				Output.SkillOutput[3].Name   :='Block';
	            Output.SkillOutput[3].ID     := 1315 ;	
				Output.SkillOutput[3].Ready  := FALSE ;
				Output.SkillOutput[3].Dummy  := FALSE ; 
	            Output.SkillOutput[3].Done   := FALSE ;
				Output.SkillOutput[3].Busy   := FALSE ;
				Output.SkillOutput[3].ParameterOutput[1].Name := 'TaskID';
				Output.SkillOutput[3].ParameterOutput[1].Dummy:= FALSE;
				Output.SkillOutput[3].ParameterOutput[1].Required:= TRUE ;
				Output.SkillOutput[3].ParameterOutput[1].MinValue:= 1;
				Output.SkillOutput[3].ParameterOutput[1].MaxValue:=30000 ;
				
				// SKILL 4 unblock INTIALISIEREN 
				
				Output.SkillOutput[4].Name   :='Unblock' ;
	            Output.SkillOutput[4].ID     := 1316 ;	
				Output.SkillOutput[4].Ready  := FALSE ;
				Output.SkillOutput[4].Dummy  := FALSE ; 
	            Output.SkillOutput[4].Done   := FALSE ;
				Output.SkillOutput[4].Busy   := FALSE ;
				Output.SkillOutput[4].ParameterOutput[1].Name :=   'TaskID';
				Output.SkillOutput[4].ParameterOutput[1].Dummy:= FALSE;
				Output.SkillOutput[4].ParameterOutput[1].Required:= TRUE ;
				Output.SkillOutput[4].ParameterOutput[1].MinValue:= 1    ;
				Output.SkillOutput[4].ParameterOutput[1].MaxValue:= 30000 ;
				
				// SKILL 5 transport INITIALISIEREN 
				
				Output.SkillOutput[5].Name   :='Transport' ;
	            Output.SkillOutput[5].ID     := 1320 ;	
				Output.SkillOutput[5].Ready  := FALSE ;
				Output.SkillOutput[5].Dummy  := FALSE ; 
	            Output.SkillOutput[5].Done   := FALSE ;
				Output.SkillOutput[5].Busy   := FALSE ;
				Output.SkillOutput[5].ParameterOutput[1].Name := 'TargetPosition X';
				Output.SkillOutput[5].ParameterOutput[1].Dummy:= FALSE;
				Output.SkillOutput[5].ParameterOutput[1].Required:= TRUE ;
				Output.SkillOutput[5].ParameterOutput[1].MinValue:= 0    ;
				Output.SkillOutput[5].ParameterOutput[1].MaxValue:= 4000 ;
				Output.SkillOutput[5].ParameterOutput[2].Name := 'TargetPosition Z';
				Output.SkillOutput[5].ParameterOutput[2].Dummy:= FALSE;
				Output.SkillOutput[5].ParameterOutput[2].Required:= FALSE ;
				Output.SkillOutput[5].ParameterOutput[2].MinValue:= 0.0    ;
				Output.SkillOutput[5].ParameterOutput[2].MaxValue:= 90.0 ;
				Output.SkillOutput[5].ParameterOutput[2].Default:= 0.0; 
				Output.SkillOutput[5].ParameterOutput[3].Name := 'Velocity';
				Output.SkillOutput[5].ParameterOutput[3].Dummy:= FALSE;
				Output.SkillOutput[5].ParameterOutput[3].Required:= FALSE ;
				Output.SkillOutput[5].ParameterOutput[3].MinValue:= 100    ;
				Output.SkillOutput[5].ParameterOutput[3].MaxValue:= 4000 ;
				Output.SkillOutput[5].ParameterOutput[3].Default := 2000;
				Output.SkillOutput[5].ParameterOutput[4].Name := 'Acceleration';
				Output.SkillOutput[5].ParameterOutput[4].Dummy:= FALSE;
				Output.SkillOutput[5].ParameterOutput[4].Required:= FALSE ;
				Output.SkillOutput[5].ParameterOutput[4].MinValue:= 100    ;
				Output.SkillOutput[5].ParameterOutput[4].MaxValue:= 4000 ;
				
				state := 0;
				
			0: // Unreserved 
				IF AwaitingAxisCnt>0 THEN
					AwaitingAxisCnt := AwaitingAxisCnt -1;
					state := 1;				
				END_IF
			
			
	    	1:		// Unreserved
					FOR i := 0 TO SkillCnt DO 
					Output.SkillOutput[i].Ready := FALSE;
					Output.SkillOutput[i].Busy := FALSE;
					Output.SkillOutput[i].Done := FALSE;
					Output.SkillOutput[i].Error := FALSE;
					END_FOR
					
					Output.SkillOutput[1].Ready                    :=TRUE; //reserve
					Output.SkillOutput[0].Ready                    :=TRUE;
					 
	            	             
	
	             	IF Input.SkillInput[1].Execute THEN 
	                
	                	Output.SkillOutput[1].Ready := FALSE ;
						Output.SkillOutput[0].Ready := FALSE ;
						Output.SkillOutput[1].Busy  := TRUE ;
						state:=10 ;
					
					END_IF
					IF Input.SkillInput[0].Execute THEN
	                	Output.SkillOutput[0].Ready := FALSE ;
						Output.SkillOutput[1].Ready := FALSE ;
						Output.SkillOutput[0].Busy  := FALSE ;
						state:=85 ;
	                			FOR i := 1 TO Grpcnt DO
										IF Output.SkillOutput[0].Busy THEN
											state := 1;
											
										END_IF
								END_FOR
						Output.SkillOutput[0].Busy  := TRUE ;
					END_IF
				   
			10:	//Reserve			     	
					IF AwaitingReservationAxis > 0 THEN
						
						//find, which mover is next in line for reservation
						
						MoverNo := AwaitingReservationAxis;
						 
						MoverInfo[AwaitingReservationAxis].blocked := FALSE;
						
						awaitingreservationaxis := 0;
						Nextaxis := F_SetAxInSection(AwaitingReservationAxis -1);
						
						//IF MoverInterface[moverNO].Setpos = WaitingAbsPosition THEN
							state := 12;
						//END_IF
							
	             	//Set mover to reserved in Global Mover Info
						
					
					
	            		MoverInfo[MoverNo].reserved:=TRUE;
						MoverInfo[MoverNo].TaskID	:= REAL_TO_INT (Input.SkillInput[1].ParameterInput[1].Value);
	                
	                	
						Output.SkillOutput[1].Done := TRUE;
						Output.SkillOutput[1].Busy := FALSE;
						Output.SkillOutput[1].Error := FALSE;
						
						
						state:=13 ;
						fbTransport(execute := FALSE, reset := TRUE); 
					END_IF
			13:		//IF NOT MoverInfo[Nextaxis].reserved THEN
					//AwaitingReservationAxis := nextaxis;
					//END_IF


					// internal Block mover next in line
					//MoverInfo[nextaxis].blocked := TRUE;
					
					IF MoverInterface[moverno].Setpos = WaitingAbsPosition	THEN		
						fbTransport( axisno := moverno, execute := TRUE,RequestPosition := F_SetInSection(WaitingAbsPosition + 2* couplegap + 5.0),requestvelo := defaultvelo);
						state := 14;
						
					ELSE
						state := 15;
					END_IF
			14: 
			
				fbTransport( axisno := moverno,RequestPosition := F_SetInSection(WaitingAbsPosition + 2* couplegap + 5.0),requestvelo := defaultvelo);
				IF fbTransport.done THEN
					state := 15;
					fbTransport(reset := TRUE);
				END_IF
		
			15:		//warten bis execute zurückgezogen
					IF NOT(Input.SkillInput[1].Execute) THEN
						Output.SkillOutput[1].Done := FALSE;
						state:=20;
					END_IF
					
					
				 
				 
	  		20:		//Reserved
					IdleTimer(IN := FALSE);
					fbIdleReservedTransport(reset := TRUE);
					state := 21;
			21:
					fbAutoBlock(axno := MoverNo);
					
					IdleTimer(IN := TRUE, PT := T#1000S);
					IF IdleTimer.Q AND (Moverinfo[F_SetAxInSection(Moverno-1)].reserved) THEN
						fbIdleReservedTransport.AxisNo := MoverNo;
						IF NOT (idletempposition = F_SetInSection( Moverinfo[F_SetAxInSection(Moverno+1)].preposition - WaySectionGap - 0.1 - Curvedistance) )THEN
						idletempposition := F_SetInSection( Moverinfo[F_SetAxInSection(Moverno+1)].preposition - WaySectionGap - 0.1 - Curvedistance);
						fbIdleReservedTransport(reset := TRUE);
						END_IF
						IF NOT F_CheckIfInCurve(idletempposition) THEN
								IF Moverinfo[F_SetAxInSection(Moverno+1)].reserved THEN
								fbIdleReservedTransport.RequestPosition := idletempposition;
								ELSE	
								fbIdleReservedTransport.RequestPosition := WaitingAbsPosition - 6 * WaySectionGap - 0.1;
								END_IF
								fbIdleReservedTransport.execute := TRUE;
								curvedistance := 0;
						ELSE
						curvedistance := curvedistance + 10.0;	
						END_IF
					END_IF
					
					fbIdleReservedTransport();
					
					FOR i := 0 TO SkillCnt DO 
					Output.SkillOutput[i].Ready := FALSE;
					Output.SkillOutput[i].Busy := FALSE;
					Output.SkillOutput[i].Done := FALSE;
					Output.SkillOutput[i].Error := FALSE;
					END_FOR
					
					Output.SkillOutput[2].Ready := TRUE;
					Output.SkillOutput[3].Ready := TRUE;
					Output.SkillOutput[5].Ready := TRUE;
					
	              	IF Input.SkillInput[5].Execute THEN 
						fbTransport(reset := TRUE);									   (*in Case of transportation*)
	                    state:=30;	
						Output.SkillOutput[5].Done := FALSE;
						Output.SkillOutput[5].Busy := TRUE;
						FOR i := 0 TO SkillCnt DO 
						Output.SkillOutput[i].Ready := FALSE;
						END_FOR					
					END_IF
	
	             	IF  Input.SkillInput[2].Execute THEN   (*Mover releasing *)
	                    state :=50;
						fbTransport(reset := TRUE);
						Output.SkillOutput[2].Busy := TRUE;
						FOR i := 0 TO SkillCnt DO 
						Output.SkillOutput[i].Ready := FALSE;
						END_FOR	
					END_IF
	
	            	IF Input.SkillInput[3].Execute THEN   (*blocking *)
	                    state:=60;
						fbTransport(reset := TRUE);
						Output.SkillOutput[3].Busy := TRUE;
						FOR i := 0 TO SkillCnt DO 
						Output.SkillOutput[i].Ready := FALSE;
						END_FOR	
				    END_IF		
	
					 
			30:	 //TRANSPORT		
					fbAutoBlock(axno := MoverNo);			
	 				IF Input.SkillInput[5].ParameterInput[4].Value> 0 AND Input.SkillInput[5].ParameterInput[4].Value < nocurvesvelo THEN
					MoverInfo[MoverNo].nocurvestop := TRUE;	
					END_IF
	                
			
			
					fbTransport(
								execute:= TRUE, 
								RequestPosition := Input.SkillInput[5].ParameterInput[1].Value,
								AxisNo:= MoverNo, 
								requestacc := Input.SkillInput[5].ParameterInput[4].Value,
								requestvelo := Input.SkillInput[5].ParameterInput[3].Value,								
								ready=> , 
								error=> , 
								busy=> , 
								done=> 
								);
	
	               IF fbTransport.done THEN             
	               state:=31 ;
				   fbTransport(reset := TRUE);
				   MoverInfo[MoverNo].blocked 	:= TRUE;				   
				   END_IF
				   
				31: 	//überprüfen ob z anforderung
						fbAutoBlock(axno := MoverNo);
						IF Input.SkillInput[5].ParameterInput[2].Value = 0 THEN
							state := 40;
						ELSE state := 32;
						END_IF
				32:		IF 		(1500<Input.SkillInput[5].ParameterInput[1].Value AND (2000+couplegap)>Input.SkillInput[5].ParameterInput[1].Value)
							OR 	(3500<Input.SkillInput[5].ParameterInput[1].Value AND (4000)>Input.SkillInput[5].ParameterInput[1].Value) OR (Input.SkillInput[5].ParameterInput[1].Value<couplegap)
							OR (0.0>Input.SkillInput[5].ParameterInput[2].Value OR 111.0<Input.SkillInput[5].ParameterInput[2].Value)
						THEN // nicht zugelassen!
							state := 41;
							fbAutoBlock(axno := MoverNo);
							Output.SkillOutput[1].done  :=FALSE;
	                    	Output.SkillOutput[2].ready :=FALSE;
	                    	Output.SkillOutput[3].ready :=FALSE;
	                    	Output.SkillOutput[4].ready :=FALSE;
	                    	Output.SkillOutput[5].done  :=FALSE;
							Output.SkillOutput[5].Error := TRUE;
							Output.SkillOutput[5].busy	:= FALSE;
						ELSE
							state := 35;				                   
						END_IF
						
						
						//z-bewegung
				35: 	fbZTransport.execute := TRUE;
						state := 36;
						
						
				36: 
						fbZTransport( zPosition := Input.SkillInput[5].ParameterInput[2].Value, axno := MoverNo);
						IF fbZTransport.done THEN						
							fbAutoBlock(execute := FALSE,axno := MoverNo);
				   			fbAutoBlock(execute := TRUE);
							state := 40;
						END_IF
						
						
				40:	    
						fbAutoBlock(axno := MoverNo,execute := FALSE);
						fbAutoBlock(axno := MoverNo,execute := TRUE);
						
						Output.SkillOutput[5].done  :=TRUE;
						Output.SkillOutput[5].busy	:= FALSE;
						
	                    state:=41;
						
						
				41:		//warten bis execute zurückgezogen
						fbAutoBlock(axno := MoverNo);
						Output.SkillOutput[5].busy	:= FALSE;
						Output.SkillOutput[5].done  :=TRUE;
							IF NOT(Input.SkillInput[5].Execute) THEN
								state:=20 ;
								Output.SkillOutput[5].Done := FALSE;
							END_IF
						
						   
				50:		//Release
							MoverInfo[MoverNo].nocurvestop := FALSE;
	              		 	MoverInfo[MoverNo].reserved := FALSE;
							MoverInfo[MoverNo].blocked := FALSE;
	                       	MoverInfo[MoverNo].TaskID	:= 0;
							MoverNo						:= 0;
							AwaitingAxisCnt := AwaitingAxisCnt +1;
							
						Output.SkillOutput[2].busy := FALSE;
						Output.SkillOutput[2].done := TRUE;
	  					state:=51 ;
						
				51:		//warten bis execute zurückgezogen
						IF NOT(Input.SkillInput[2].Execute) THEN
							state:=0 ;
							Output.SkillOutput[2].Done := FALSE;
						END_IF
						   
						//Block
				60:	  
							
	                        
						MoverInfo[MoverNo].blocked 	:= TRUE;
						  
	                    Output.SkillOutput[3].busy:=FALSE;
						Output.SkillOutput[3].done:=TRUE;
						   
	                    state:=61;
						
				61:		//warten bis execute zurückgezogen
						Output.SkillOutput[3].done:=TRUE;
						IF NOT(Input.SkillInput[3].Execute) THEN
							state:=70 ;
							Output.SkillOutput[3].Done := FALSE;
						END_IF
						   
	            70:		//BLOCKED
						FOR i := 0 TO SkillCnt DO 
						Output.SkillOutput[i].Ready := FALSE;
						Output.SkillOutput[i].Busy := FALSE;
						Output.SkillOutput[i].Done := FALSE;
						Output.SkillOutput[i].Error := FALSE;
						END_FOR			
						Output.SkillOutput[4].Ready := TRUE;
						
						IF Input.SkillInput[4].Execute THEN
							state := 80;
							Output.SkillOutput[4].busy   :=TRUE ;
							Output.SkillOutput[4].Ready := FALSE;
							
						END_IF
	
	
	           	80:         // Unblock;
						MoverInfo[MoverNo].blocked := FALSE;
						MoverInterface[Moverno].Buddyenable := FALSE;
						Output.SkillOutput[4].busy  :=FALSE ;
						Output.SkillOutput[4].Done	:= TRUE;
						
						state := 81;
						
	       		81:     //warten bis execute zurückgezogen
						Output.SkillOutput[4].Done	:= TRUE;
						IF NOT(Input.SkillInput[4].Execute) THEN
							state:=20; 
							Output.SkillOutput[4].Done := FALSE;
						END_IF       
				


				85:		//Initialization
						//IF NOT GVL.ClientExecute THEN
						InitMoverNo := AwaitingReservationAxis;
						state := 86;
						Output.SkillOutput[0].Error := FALSE;
						//END_IF
				86: 	
						state := 87;
						FOR i := 1 TO grpcnt DO
							IF MoverInfo[i].reserved THEN
								state := 86;
							END_IF
						END_FOR
						IF NOT MoverInfo[F_SetAxInSection(grp :=InitMoverNo-1)].reserved THEN
						InitMoverNo := F_SetAxInSection(InitMoverNo-1);
						ELSE
							state := 88;
						END_IF
						
				87: // alle mover unreserved
					IF NOT (AwaitingReservationAxis = 0) THEN
					InitMoverNo := F_SetAxInSection(grp := AwaitingReservationAxis +1);
					state := 88;
					Timeout(IN := FALSE);
					END_IF
					
				88: //OPC COnnection
					//IF NOT GVL.ClientExecute THEN
							AveragedPosition := 0;
							ClientWrite := FALSE;
							FOR i := 1 TO 10 DO Gvl.MeasuredPosition[i] := 0;
								
							END_FOR
								
							GVL.ClientExecute := TRUE;
							GVL.ClientModuleServerUrl 	:= Input.SkillInput[0].ParameterInput[0].StringValue;
							GVL.ClientReadIdentifier	:= Input.SkillInput[0].ParameterInput[1].StringValue;
							GVL.ClientWriteIdentifier 	:= Input.SkillInput[0].ParameterInput[2].StringValue;
							GVL.ClientNamespaceIndex	:= STRING_TO_UINT (Input.SkillInput[0].ParameterInput[3].StringValue);
							GVL.ClientNamespaceUri		:= Input.SkillInput[0].ParameterInput[4].StringValue;
							IF GVL.ClientReadEstablished THEN
								state := 89;
							END_IF
							
							Timeout(IN := TRUE, PT := T#10S);
							IF Timeout.Q THEN
								Timeout(IN := FALSE);
							state := 107;
							Output.SkillOutput[0].Busy := FALSE;
							Output.SkillOutput[0].Error := TRUE;
								
							END_IF
					//END_IF
					
				89: MoverInfo[InitMoverNo].reserved := TRUE;
					fbTransport(execute := TRUE, AxisNo := InitMoverNo,RequestPosition := F_SetInSection(WaitingAbsPosition - 5.5* WaySectionGap), requestvelo := maxvelo);
					IF MoverInterface[InitMoverNo].Targetpos = F_SetInSection(WaitingAbsPosition - 5.5* WaySectionGap) THEN
                  		state := 90;
					END_IF
				90: fbTransport();
					IF fbTransport.done THEN
						state := 91;
						fbTransport(reset := TRUE);
					END_IF
				91:	
					fbTransport(execute := TRUE, AxisNo := InitMoverNo,RequestPosition := WaitingAbsPosition + 2.5* WaySectionGap, requestvelo := initvelo);
					IF MoverInterface[InitMoverNo].Targetpos = WaitingAbsPosition + 2.5* WaySectionGap THEN
                  		state := 92;
					END_IF
					
				
				92: fbTransport(); // erste suche
					IF bInput THEN 
					tempposition := F_SetInSection(ax[InitMoverNo*2].NcToPlc.ModuloActPos );
					fbTransport(execute := FALSE, reset := TRUE);
					state := 95;
					END_IF
					IF fbTransport.done THEN
						IF measuredposition[1] = 0 THEN
							state := 106;
						ELSE
						state := 95;
						END_IF
					END_IF
				
					
				95: IF measuredcycles = measurementCycles THEN
						state  := 100;
					ELSE					
					//in position fahren
					fbTransport(execute := TRUE, AxisNo := InitMoverNo, RequestPosition := F_SetInSection(Tempposition + ((EXPT(-1,measuredcycles)) * 100)),requestvelo := 2000);
					IF NOT bInput AND fbTransport.done THEN
						
					state := 96;
					END_IF
					END_IF
					
				96: //Messung
					fbTransport(execute := TRUE, AxisNo := InitMoverNo, RequestPosition := F_SetInSection(Tempposition - ((EXPT(-1,measuredcycles)) * 300)) ,requestvelo := 50);
					IF bInput THEN
					MeasuredPosition[measuredcycles +1] := ax[2*InitMoverNo].NcToPlc.ModuloActPos;
					measuredcycles := measuredcycles +1;
					fbTransport(execute := FALSE, Reset := TRUE);
					state := 95;
					END_IF
					IF fbTransport.done THEN
						state := 95;
						repeatcounter := repeatcounter + 1;
					END_IF
					IF Repeatcounter > Measurementcycles + 20 THEN
						
							state := 107;
							Output.SkillOutput[0].Busy := FALSE;
							Output.SkillOutput[0].Error := TRUE;
							
					END_IF
					
				100: 
						i := 1;
						state := 103;
				103: 
					IF i <= measurementCycles THEN
						AveragedPosition := AveragedPosition + (EXPT(measurementCycles,-1) * ( measuredposition[i]));
						i := i+1;
					ELSE
						fbTransport(reset := TRUE, execute := FALSE);
						state := 105;
						Timeout(IN := FALSE);
						AveragedPosition := F_SetInSection(AveragedPosition - 33.5);					
					END_IF
				105: 
					fbTransport(execute := TRUE, AxisNo := InitMoverNo, RequestPosition := AveragedPosition);
					IF fbTransport.done THEN
						state := 106;
						Timeout(IN := FALSE);
						fbTransport(reset := TRUE);
					END_IF
				106: 	ClientWrite := TRUE;
						Timeout(IN := TRUE, PT := T#100S);
							IF Timeout.Q THEN
								Timeout(IN := FALSE);
							state := 1070;
							Output.SkillOutput[0].Busy := FALSE;
							Output.SkillOutput[0].Error := TRUE;
								
							END_IF
						IF GVL.ClientDone THEN
						
					 	state := 107;
						OUTput.SkillOutput[0].Done := TRUE;
						OUTput.SkillOutput[0].busy := FALSE; 
					 	END_IF
			    107:	//auf execute zurückziehen warten 
						ClientExecute := FALSE;
						fbTransport(reset := TRUE);
						IF NOT Input.SkillInput[0].Execute THEN
						MoverInfo[InitMoverNo].reserved := FALSE;
						OUTput.SkillOutput[0].Done := FALSE;
						Output.SkillOutput[0].Busy := FALSE;
						state := 1;
						measuredcycles := 0;
						repeatcounter := 0;
						END_IF
					
					 
							  
						
	END_CASE
	
ELSE //SUPPRESSED!
	fbSuppressedTransport(
	surpressall := TRUE,	
	execute:= TRUE, 
	RequestPosition:= MoverInfo[MoverNo].SurpressedPosition, 
	AxisNo:= MoverNo, 
	ready=> , 
	error=> , 
	busy=> , 
	done=> );
	IF fbSuppressedTransport.done THEN
		fbTransport.reset := TRUE;
		MoverInfo[MoverNo].surpressed := FALSE;
				
	END_IF
END_IF

ELSE
	IF restartstate = 2 THEN
		state := 0;
		fbTransport(reset := TRUE);
		restartstate := 3;
		moverno := 0;
	END_IF
END_IF

Output.ConnectionTestOutput := INput.ConnectionTestInput;

END_FUNCTION_BLOCK

// ---- POUs/SkillHandle/FB_Transport.TcPOU
FUNCTION_BLOCK FB_Transport
VAR_INPUT
	execute: BOOL;
	RequestPosition: LREAL;
	AxisNo: INT;
	reset: BOOL;
	requestvelo: LREAL;
	requestacc: LREAL;
	surpressall: BOOL;
	test1: BOOL;
	test2: BOOL;
END_VAR
VAR_OUTPUT
	ready: BOOL;
	error: BOOL;
	busy: BOOL;
	done: BOOL;
END_VAR
VAR
	///FBs
	calculateWaysection: FB_CalculateWaysection;
	checkWaysection: FB_CheckWaysection;
	Clockwise: BOOL;
	TempPreposition: LREAL;
	TempPostposition: LREAL;
	BlockingAxisNo: INT;
	state: INT := 10;
	surpressCheck	: BOOL := FALSE;
	i: INT;
	CatchUp	: BOOL;
END_VAR

IF reset THEN
	state := 10;
	reset := FALSE;
	done := FALSE;
	execute := FALSE;
	calculateWaysection(Execute := FALSE);
	checkWaysection(Execute := FALSE);
END_IF
IF execute THEN 
	done := FALSE;
	busy := TRUE;
	CASE state OF 
	10: // calculate clockwise
			calculateWaysection(
					Clockwise:= TRUE, 
					Startpos:= MoverInterface[AxisNo].Setpos,
					Endpos:= RequestPosition, 
					WaySectionGap:= WaySectionGap, 
					Execute:= TRUE, 
					Prepos=> TempPreposition, 
					Postpos=> TempPostposition, 
					done=> );
			IF calculateWaysection.done THEN state := 15; END_IF
			
	15: // immer nur einer gleichzeitig checken:
		IF Reservingaxis = 0  OR Reservingaxis = AxisNo THEN
			Reservingaxis := AxisNo;
			state := 20;
		END_IF
	20: // check clockwise waysection & reserve if free
			checkWaysection(
							CheckPreposition:= TempPreposition, 
							CheckPostposition:= TempPostposition, 
							CheckMoverNo:= AxisNo , 
							Execute:= TRUE, 
							SectionFree=> , 
							axisblocking=> , 
							done=> );
							
			IF checkWaysection.done THEN
				Reservingaxis := 0;
					IF checkWaysection.SectionFree THEN
						//Section frei -> Reservieren!
							MoverInfo[AxisNo].postposition 	:= TempPostposition;
							MoverInfo[AxisNo].preposition	:= TempPreposition;
							state := 100;
							Clockwise := TRUE;
							
						ELSE
							state := 25;
					END_IF
				
			END_IF
	
	25: // immer nur einer gleichzeitig checken:
		IF Reservingaxis = 0 OR Reservingaxis = AxisNo THEN
			Reservingaxis := AxisNo;
			state := 30;
		END_IF	
	
	30: //calculate counter-clockwise
		calculateWaysection(
					Clockwise:= FALSE, 
					Startpos:= MoverInterface[AxisNo].Setpos,
					Endpos:= RequestPosition, 
					WaySectionGap:= WaySectionGap, 
					Execute:= TRUE, 
					Prepos=> TempPreposition, 
					Postpos=> TempPostposition, 
					done=> );
			IF calculateWaysection.done THEN state := 40; END_IF
	
	40: //check counter-clockwise waysection
		checkWaysection(
							CheckPreposition:= TempPreposition, 
							CheckPostposition:= TempPostposition, 
							CheckMoverNo:= AxisNo , 
							Execute:= TRUE, 
							SectionFree=> , 
							axisblocking=> , 
							done=> );
							
			IF checkWaysection.done THEN
				Reservingaxis := 0;
					IF checkWaysection.SectionFree
						THEN //Section frei -> Reservieren!
							MoverInfo[AxisNo].postposition 	:= TempPostposition;
							MoverInfo[AxisNo].preposition	:= TempPreposition;
							state := 100;
							Clockwise := FALSE;
					ELSE	//section nicht frei
						state := 50;
					END_IF			
			END_IF
	
	50: //Find Out blocking axNo
		BlockingAxisNo := AxisNo -1;
		IF AxisNo = 1 THEN
			BlockingAxisNo := grpcnt;
		END_IF
		state := 60;
	
	60: 		test1 :=F_CheckIfInSection(Position := WaitingAbsPosition - 6 * WaySectionGap, postposition := MoverInterface[AxisNo].Setpos, preposition := F_SetInSection(TempPreposition - WaySectionGap -0.1));
				test2 := F_CheckSurpressedSection(SurpressedPosition := F_SetInSection(TempPreposition - WaySectionGap -0.1), preposition := F_SetInSection(WaitingAbsPosition - 3 * couplegap), postposition := MoverInterface[AxisNo].Setpos);
		IF NOT surpressCheck THEN
			state  := 10;
			surpresscheck := TRUE;
		ELSE
			
				IF 
					NOT MoverInfo[BlockingAxisNo].blocked 
					AND NOT (Moverinfo[axisno].surpressed AND Moverinfo[F_SetAxInSection(axisno +1)].surpressed )    
					AND 	(surpressall OR
							(*  (NOT F_CheckIfInSection(Position:=MoverInterface[blockingaxisno].Targetpos, postposition := WaitingAbsPosition, preposition := F_SetInSection( Waitingabsposition - 6 * (waysectiongap + 0.1))) 
								AND NOT F_CheckSurpressedSection(SurpressedPosition := F_SetInSection(TempPreposition - WaySectionGap -0.1), preposition := F_SetInSection(WaitingAbsPosition - 3 * couplegap), postposition := MoverInterface[AxisNo].Setpos))
							*)
							NOT F_CheckIfInSection(Position := WaitingAbsPosition - 6 * WaySectionGap, postposition := MoverInterface[AxisNo].Setpos, preposition := F_SetInSection(TempPreposition - WaySectionGap -0.2))
							)
						
							// ACHSE Verdrängen
				THEN	MoverInfo[BlockingAxisNo].surpressed := TRUE;
						surpresscheck := FALSE;	
							//verdängungsposition berechnen
							IF NOT (F_CheckIfInCurve (TempPreposition - WaySectionGap -0.2) AND MoverInfo[i].nocurvestop) THEN
							MoverInfo[BlockingAxisNo].SurpressedPosition :=  F_SetInSection(TempPreposition - WaySectionGap -0.2);
							ELSE
								IF F_SetInSection(TempPreposition - WaySectionGap -0.2 ) > 2500 THEN
									// hintere kurve
									MoverInfo[BlockingAxisNo].SurpressedPosition :=  3450;
								ELSE
									//vordere Kurve
									MoverInfo[BlockingAxisNo].SurpressedPosition :=  1450;
								END_IF
							
							END_IF
							
							
							//gegen den uhrzeigersinn ausweichen:
							MoverInfo[BlockingAxisNo].SupressedClockwise := FALSE;
							state := 70; //auf verdrängung warten
					ELSE
							state := 10; //warten/neue Berechnung
							IF (Moverinfo[axisno].surpressed AND Moverinfo[F_SetAxInSection(axisno +1)].surpressed ) THEN
							ADSLOGSTR(ADSLOG_MSGTYPE_HINT, 'trying to surpress all movers! Help!', '');
							state := 10;	
							END_IF
				END_IF
			END_IF
	
	70: 	//Wait untill suppressed movement done
			// Supressed mover Rücken auf
			
			IF  (MoverInfo[AxisNo].preposition - MoverInfo[BlockingAxisNo].postposition ) > (surpressinggap + 600) THEN
				
			
			MoverInfo[AxisNo].preposition 	:= F_SetinSection(MoverInfo[BlockingAxisNo].postposition + surpressinggap);
			MoverInfo[AxisNo].postposition	:= F_SetinSection(MoverInterface[AxisNo].Setpos + waysectiongap);
			MoverInterface[AxisNo].targetpos := F_SetInSection(MoverInfo[BlockingAxisNo].postposition + waysectiongap + surpressinggap);
			CAInterface.MoverInterface[AxisNo].Clockwise := FALSE;
			CatchUp := TRUE;
			ELSE
			CatchUp := FALSE;
			END_IF
			surpresscheck := FALSE;
				
			state := 71;
	71: 	
			// immer nur einer gleichzeitig checken:
			IF Reservingaxis = 0 OR Reservingaxis = AxisNo THEN
				Reservingaxis := AxisNo;
				state := 30;
			END_IF	
	72:
			checkWaysection(
							CheckPreposition:= TempPreposition, 
							CheckPostposition:= TempPostposition, 
							CheckMoverNo:= AxisNo , 
							Execute:= TRUE, 
							SectionFree=> , 
							axisblocking=> , 
							done=> );
			
							
			IF checkWaysection.done THEN
					Reservingaxis := 0;
					IF checkWaysection.SectionFree
						THEN //Section frei -> Reservieren!
							MoverInfo[AxisNo].postposition 	:= TempPostposition;
							MoverInfo[AxisNo].preposition	:= TempPreposition;
							state := 100;
							Clockwise := FALSE;
					ELSE
						state :=71;
					END_IF			
			END_IF
			IF CatchUp THEN
				//reservierten bereich während der fahr freigeben
			IF ((CAInterface.MoverInterface[axisno].Setpos + WaySectionGap)> railLength) THEN //bereich überprüfen
						MoverInfo[AxisNo].postposition := CAInterface.MoverInterface[axisno].Setpos + WaySectionGap -railLength;
			ELSE
						MoverInfo[AxisNo].postposition := CAInterface.MoverInterface[axisno].Setpos + WaySectionGap;
			END_IF
			state := 70;
			END_IF
	
		///BEWEGUNGSAUSFÜHRUNG
	100: 	CAInterface.MoverInterface[AxisNo].Targetpos := RequestPosition;
			CAInterface.MoverInterface[AxisNo].Clockwise := Clockwise;
			CAInterface.MoverInterface[AxisNo].MovementDone := FALSE;
			IF (requestacc > 0.0 AND requestacc < maxacc) THEN
			CAInterface.MoverInterface[AxisNo].Acceleration := requestacc;
			ELSE 
				CAInterface.MoverInterface[AxisNo].Acceleration := defaulacc;
			END_IF
			IF (requestvelo > 0.0 AND requestvelo < maxvelo) THEN
			CAInterface.MoverInterface[AxisNo].Velocity := requestvelo;
			ELSE 
				CAInterface.MoverInterface[AxisNo].Velocity := defaultvelo;
			END_IF
			surpresscheck := FALSE;	
			state := 101;
			
	101:	//reservierten bereich während der fahrt freigeben
			IF Clockwise 
			THEN 
				// Preposition aktualisieren
				
					IF ((CAInterface.MoverInterface[axisno].Setpos - WaySectionGap)< 0.0) THEN //bereich überprüfen
						MoverInfo[AxisNo].preposition := CAInterface.MoverInterface[axisno].Setpos - WaySectionGap +railLength;
					ELSE
						MoverInfo[AxisNo].preposition := CAInterface.MoverInterface[axisno].Setpos - WaySectionGap;
					END_IF
				
			ELSE
				//Postposition aktualisieren
					IF ((CAInterface.MoverInterface[axisno].Setpos + WaySectionGap)> railLength) THEN //bereich überprüfen
						MoverInfo[AxisNo].postposition := CAInterface.MoverInterface[axisno].Setpos + WaySectionGap -railLength;
					ELSE
						MoverInfo[AxisNo].postposition := CAInterface.MoverInterface[axisno].Setpos + WaySectionGap;
					END_IF
			END_IF
			
			//Auf Ende Warten
			IF CAInterface.MoverInterface[AxisNo].MovementDone THEN
		
				state :=  10;
				execute := FALSE;
				busy := FALSE;
				done := TRUE;
					// letztes mal pre/post aktuallisieren
								IF Clockwise 
								THEN 
									// Preposition aktualisieren
									
										IF ((CAInterface.MoverInterface[axisno].Setpos - WaySectionGap)< 0.0) THEN //bereich überprüfen
											MoverInfo[AxisNo].preposition := CAInterface.MoverInterface[axisno].Setpos - WaySectionGap +railLength;
										ELSE
											MoverInfo[AxisNo].preposition := CAInterface.MoverInterface[axisno].Setpos - WaySectionGap;
										END_IF
									
								ELSE
									//Postposition aktualisieren
										IF ((CAInterface.MoverInterface[axisno].Setpos + WaySectionGap)> railLength) THEN //bereich überprüfen
											MoverInfo[AxisNo].postposition := CAInterface.MoverInterface[axisno].Setpos + WaySectionGap -railLength;
										ELSE
											MoverInfo[AxisNo].postposition := CAInterface.MoverInterface[axisno].Setpos + WaySectionGap;
										END_IF
								END_IF
			END_IF
	
	
	
		
	END_CASE
	ELSE state := 10;
END_IF

END_FUNCTION_BLOCK

// ---- POUs/SkillHandle/F_CheckIfInSection.TcPOU
FUNCTION F_CheckIfInSection : BOOL
VAR_INPUT
	Position: LREAL;
	postposition: LREAL;
	preposition: LREAL;
END_VAR
VAR
	InSection: BOOL;
END_VAR


	InSection := FALSE;
		IF postposition>preposition 
		THEN
				//DER RESERVIERTE BEREICH GEHT NICHT ÜBER NULL:	
					
					// gesamter bereich umschlungen?
					IF Position >  preposition AND Position <= PostPosition THEN
						InSection:= TRUE;
					END_IF
				
		ELSE
				//DER RESERVIERTE BEREICH GEHT ÜBER NULL!
				//Bereich 1: 0 bis Postpos:
					// Grenze in Bereich?
					IF((Position>=0.0) AND (Position<=postposition)) 
						THEN 
							InSection:= TRUE;
								
					END_IF
				
				//Bereich 2: Prepos bis 4000
					// Grenze in Bereich?
					IF((Position>=preposition) AND (Position<=raillength)) 
						THEN 
							InSection:= TRUE;
					END_IF	
		END_IF

F_CheckIfInSection := inSection;

END_FUNCTION

// ---- POUs/SkillHandle/F_SetInSection.TcPOU
FUNCTION F_SetInSection : LREAL
VAR_INPUT
	Position: LREAL;
END_VAR
VAR
	output: LREAL;
END_VAR

IF (Position >= raillength) THEN
	output := position -raillength;
ELSE
	IF (Position < 0.0) THEN
		output := position + raillength;
	ELSE
	output := Position;
	END_IF
END_IF
F_SetInSection := output;

END_FUNCTION

// ---- POUs/SkillHandle/F_CheckSurpressedSection.TcPOU
FUNCTION F_CheckSurpressedSection : BOOL
VAR_INPUT
	SurpressedPosition: LREAL;
	postposition: LREAL;
	preposition: LREAL;
END_VAR
VAR
	InSection: BOOL;
END_VAR


	InSection := FALSE;
		IF postposition>preposition 
		THEN
				//DER RESERVIERTE BEREICH GEHT NICHT ÜBER NULL:	
					
					// gesamter bereich umschlungen?
					IF SurpressedPosition >  preposition AND SurpressedPosition <= PostPosition THEN
						InSection:= TRUE;
					END_IF
				
		ELSE
				//DER RESERVIERTE BEREICH GEHT ÜBER NULL!
				//Bereich 1: 0 bis Postpos:
					// Grenze in Bereich?
					IF((SurpressedPosition>=0.0) AND (SurpressedPosition<=postposition)) 
						THEN 
							InSection:= TRUE;
								
					END_IF
				
				//Bereich 2: Prepos bis 4000
					// Grenze in Bereich?
					IF((SurpressedPosition>=preposition) AND (SurpressedPosition<=raillength)) 
						THEN 
							InSection:= TRUE;
					END_IF	
		END_IF

F_CheckSurpressedSection := inSection;

END_FUNCTION

// ---- POUs/SkillHandle/F_SetAxInSection.TcPOU
FUNCTION F_SetAxInSection : INT
VAR_INPUT
	grp: INT := 0;
END_VAR

IF grp < 1 THEN 
	F_SetAxInSection := grp + grpcnt;
ELSE
	IF grp > grpcnt THEN
		F_SetAxInSection := grp  - grpcnt;
	ELSE
		F_SetAxInSection := grp;
	END_IF
END_IF

END_FUNCTION

// ---- POUs/SkillHandle/F_CheckIfInCurve.TcPOU
FUNCTION F_CheckIfInCurve : BOOL
VAR_INPUT
	Position: LREAL;
END_VAR
VAR
	pre1: LREAL := 1490.0;
	end1: LREAL := 2010.0;
	
	pre2: LREAL := 3490.0;
	
	end2: LREAL := 10.0;
END_VAR

F_CheckIfInCurve := F_CheckIfInSection(Position := Position, postposition := end1, preposition := pre1) or F_CheckIfInSection(Position := Position, postposition := end2, preposition := pre2);

END_FUNCTION

// ---- POUs/SkillHandle/FB_AutoBlock.TcPOU
FUNCTION_BLOCK FB_AutoBlock
VAR_INPUT
	execute: BOOL;
	axno: INT;
	blockingtime: TIME := TIME#2s0ms;
END_VAR
VAR
	state: INT := 0;
	fbTimer: TON;
END_VAR

IF NOT Execute THEN
	state := 0;
ELSE
	CASE state OF
		
	0: 
		MoverInfo[axno].blocked := TRUE;
		fbTimer(IN := FALSE);
		fbTimer(IN := TRUE, PT := blockingtime);
		state := 1;
	1:	
		fbTimer();
		IF fbTimer.Q THEN
			MoverInfo[axno].blocked := FALSE;
			execute := FALSE;
			state := 0;
		END_IF
		
	
	
	
	
	END_CASE
END_IF

END_FUNCTION_BLOCK

// ---- POUs/SkillHandle/FB_ZTransport.TcPOU
FUNCTION_BLOCK FB_ZTransport
VAR_INPUT
	execute: BOOL;
	axno: INT;
	zPosition: LREAL;
END_VAR
VAR_OUTPUT
	done: BOOL;
	busy: BOOL;
	error: BOOL;
END_VAR
VAR
	state: INT := 0;
	gap: LREAL;
END_VAR

IF execute THEN
	done	:= FALSE;/// 
	busy := TRUE; ///
	CASE state OF
		
	0: //gap berechnen 12 30 154
		done	:= FALSE;
		busy := TRUE;
		gap := (-0.4123*zPosition)+ zerohightdistance;
		state := 5;
		
	5:	
		CAInterface.MoverInterface[axno].Buddyenable := FALSE;
		IF NOT CAInterface.MoverInterface[axno].Buddyactive THEN
			state := 10;
		END_IF
		
	10: 
		// an CA übergeben
		CAInterface.MoverInterface[axno].Buddygap := gap;
		CAInterface.MoverInterface[axno].Buddyenable := TRUE;
		state := 20;

	20: 
		IF  CAInterface.MoverInterface[axno].Buddyactive THEN
		done := TRUE;
		busy := FALSE;
		execute := FALSE;
		state := 0;
		END_IF
	
	
	
	END_CASE
END_IF

END_FUNCTION_BLOCK

// ---- POUs/SkillHandle/FB_FreeTransport.TcPOU
FUNCTION_BLOCK FB_FreeTransport
VAR_INPUT
	execute: BOOL;
	RequestPosition: LREAL;
	AxisNo: INT;
	reset: BOOL;
END_VAR
VAR_OUTPUT
	ready: BOOL;
	error: BOOL;
	busy: BOOL;
	done: BOOL;
END_VAR
VAR
	///FBs
	calculateWaysection: FB_CalculateWaysection;
	checkWaysection: FB_CheckWaysection;
	Clockwise: BOOL;
	TempPreposition: LREAL;
	TempPostposition: LREAL;
	BlockingAxisNo: INT;
	PostmoverNo: INT;
	state: INT := 10;
	i: INT;
	fbSuppressedTransport: FB_Transport;
END_VAR

//Nummer des nächsten Movers herausfinden
PostmoverNo := F_SetAxInSection( AxisNo +1);


IF NOT Restart THEN

IF NOT MoverInfo[AxisNo].surpressed THEN
	

			IF execute THEN 
				MoverInterface[axisno].Buddyenable:= FALSE;
				done := FALSE;
				busy := TRUE;
				CASE state OF 
				10: // calculate counter-clockwise
						calculateWaysection(
								Clockwise:= FALSE, 
								Startpos:= MoverInterface[AxisNo].Setpos,
								Endpos:= RequestPosition, 
								WaySectionGap:= WaySectionGap, 
								Execute:= TRUE, 
								Prepos=> TempPreposition, 
								Postpos=> TempPostposition, 
								done=> );
						IF calculateWaysection.done THEN state := 15; END_IF
				15:  // immer nur einer gleichzeitig checken:
						IF Reservingaxis = 0 OR Reservingaxis = AxisNo THEN
							Reservingaxis := AxisNo;
							state := 20;
						END_IF
				20: // check counter-clockwise waysection & reserve if free
						checkWaysection(
										CheckPreposition:= TempPreposition, 
										CheckPostposition:= TempPostposition, 
										CheckMoverNo:= AxisNo , 
										Execute:= TRUE, 
										SectionFree=> , 
										axisblocking=> , 
										done=> );
										
						IF checkWaysection.done THEN
							Reservingaxis := 0;
								IF checkWaysection.SectionFree
									THEN //Section frei -> Reservieren!
										MoverInfo[AxisNo].postposition 	:= TempPostposition;
										MoverInfo[AxisNo].preposition	:= TempPreposition;
										state := 100;
										Clockwise := FALSE;
								ELSE state := 25;
								END_IF
							
						END_IF
				
				25: // immer nur einer gleichzeitig checken:
					IF Reservingaxis = 0 OR Reservingaxis = AxisNo THEN
						Reservingaxis := AxisNo;
						state := 30;
					END_IF		
				
				30: //calculate clockwise
					calculateWaysection(
								Clockwise:= TRUE, 
								Startpos:= MoverInterface[AxisNo].Setpos,
								Endpos:= RequestPosition, 
								WaySectionGap:= WaySectionGap, 
								Execute:= TRUE, 
								Prepos=> TempPreposition, 
								Postpos=> TempPostposition, 
								done=> );
						IF calculateWaysection.done THEN state := 40; END_IF
				
				40: //check clockwise waysection
					checkWaysection(
										CheckPreposition:= TempPreposition, 
										CheckPostposition:= TempPostposition, 
										CheckMoverNo:= AxisNo , 
										Execute:= TRUE, 
										SectionFree=> , 
										axisblocking=> , 
										done=> );
										
						IF checkWaysection.done THEN
							Reservingaxis := 0;
								IF checkWaysection.SectionFree
									THEN //Section frei -> Reservieren!
										MoverInfo[AxisNo].postposition 	:= TempPostposition;
										MoverInfo[AxisNo].preposition	:= TempPreposition;
										state := 100;
										Clockwise := TRUE;
								ELSE	//section nicht frei
									state := 50;
								END_IF			
						END_IF
				
						
				50: //Aufschließen
					calculateWaysection(
								Clockwise:= TRUE, 
								Startpos:= MoverInterface[AxisNo].Setpos,
								Endpos:= F_SetInSection(Position := (MoverInfo[PostmoverNo].preposition - WaySectionGap - 0.1)) , 
								WaySectionGap:= WaySectionGap, 
								Execute:= TRUE, 
								Prepos=> TempPreposition, 
								Postpos=> TempPostposition, 
								done=> );
						IF calculateWaysection.done THEN state := 55; END_IF
						
				55:		IF Reservingaxis = 0 THEN
						Reservingaxis := AxisNo;
						state := 60;
						END_IF
						
				60:		
						checkWaysection(
										CheckPreposition:= TempPreposition, 
										CheckPostposition:= TempPostposition, 
										CheckMoverNo:= AxisNo , 
										Execute:= TRUE, 
										SectionFree=> , 
										axisblocking=> , 
										done=> );
										
						IF checkWaysection.done THEN
								Reservingaxis := 0;
								IF checkWaysection.SectionFree
									THEN //Section frei -> Reservieren!
										MoverInfo[AxisNo].postposition 	:= TempPostposition;
										MoverInfo[AxisNo].preposition	:= TempPreposition;
										state := 70;
										Clockwise := TRUE;
								ELSE	//section nicht frei
									state := 10;
								END_IF			
						END_IF
						
				70: 	CAInterface.MoverInterface[AxisNo].Targetpos := F_SetInSection(MoverInfo[PostmoverNo].preposition - WaySectionGap - 0.1);
						CAInterface.MoverInterface[AxisNo].Clockwise := Clockwise;
						CAInterface.MoverInterface[AxisNo].MovementDone := FALSE;
						CAInterface.MoverInterface[AxisNo].Velocity := freevelo;
						CAInterface.MoverInterface[AxisNo].Acceleration := freeacc;
						state := 71;
						
				71:	//reservierten bereich während der fahrt freigeben
						IF Clockwise 
						THEN 
							// Preposition aktualisieren
							
								IF ((CAInterface.MoverInterface[axisno].Setpos - WaySectionGap)< 0.0) THEN //bereich überprüfen
									MoverInfo[AxisNo].preposition := CAInterface.MoverInterface[axisno].Setpos - WaySectionGap +railLength;
								ELSE
									MoverInfo[AxisNo].preposition := CAInterface.MoverInterface[axisno].Setpos - WaySectionGap;
								END_IF
							
						ELSE
							//Postposition aktualisieren
								IF ((CAInterface.MoverInterface[axisno].Setpos + WaySectionGap)> railLength) THEN //bereich überprüfen
									MoverInfo[AxisNo].postposition := CAInterface.MoverInterface[axisno].Setpos + WaySectionGap -railLength;
								ELSE
									MoverInfo[AxisNo].postposition := CAInterface.MoverInterface[axisno].Setpos + WaySectionGap;
								END_IF
						END_IF
						
						//Auf Ende Warten
						IF CAInterface.MoverInterface[AxisNo].MovementDone THEN
					
							state :=  10;
						ELSE
							state := 30;	
						END_IF
				
					///BEWEGUNGSAUSFÜHRUNG
				100: 	CAInterface.MoverInterface[AxisNo].Targetpos := RequestPosition;
						CAInterface.MoverInterface[AxisNo].Clockwise := Clockwise;
						
						CAInterface.MoverInterface[AxisNo].MovementDone := FALSE;
						CAInterface.MoverInterface[AxisNo].Acceleration := freeacc;
						CAInterface.MoverInterface[AxisNo].Velocity := freevelo;
						
						state := 101;
						
				101:	//reservierten bereich während der fahrt freigeben
						IF Clockwise 
						THEN 
							// Preposition aktualisieren
							
								IF ((CAInterface.MoverInterface[axisno].Setpos - WaySectionGap)< 0.0) THEN //bereich überprüfen
									MoverInfo[AxisNo].preposition := CAInterface.MoverInterface[axisno].Setpos - WaySectionGap +railLength;
								ELSE
									MoverInfo[AxisNo].preposition := CAInterface.MoverInterface[axisno].Setpos - WaySectionGap;
								END_IF
							
						ELSE
							//Postposition aktualisieren
								IF ((CAInterface.MoverInterface[axisno].Setpos + WaySectionGap)> railLength) THEN //bereich überprüfen
									MoverInfo[AxisNo].postposition := CAInterface.MoverInterface[axisno].Setpos + WaySectionGap -railLength;
								ELSE
									MoverInfo[AxisNo].postposition := CAInterface.MoverInterface[axisno].Setpos + WaySectionGap;
								END_IF
						END_IF
						
						//Auf Ende Warten
						IF CAInterface.MoverInterface[AxisNo].MovementDone THEN
					
							state :=  10;
							execute := FALSE;
							busy := FALSE;
							done := TRUE;
						END_IF
				
						
				
					
				END_CASE
			END_IF
ELSE //suppressed!
	fbSuppressedTransport(
	surpressall := TRUE,
	execute:= TRUE, 
	RequestPosition:= MoverInfo[AxisNo].SurpressedPosition, 
	AxisNo:= AxisNo, 
	requestvelo := freevelo,
	ready=> , 
	error=> , 
	busy=> , 
	done=> );
	IF fbSuppressedTransport.done THEN
		state := 10;
		MoverInfo[AxisNo].surpressed := FALSE;
				
	END_IF

END_IF

ELSE
	IF restartstate = 3 THEN
		state := 10;
		restartstate := 4;
	END_IF
END_IF

END_FUNCTION_BLOCK

// ---- POUs/SkillHandle/FB_FreeSlotHandle.TcPOU
FUNCTION_BLOCK FB_FreeSlotHandle
VAR_INPUT
	autoexecute: BOOL;
END_VAR
VAR
	fbFreeTransport: ARRAY[1..grpcnt] OF FB_FreeTransport;
	i: INT;
	initdone: BOOL;
	initax: INT := 3;
	minposition: LREAL := 4000.0;
END_VAR

IF NOT initdone AND((MoverInterface[1].MovementDone) AND (MoverInterface[2].MovementDone) AND (MoverInterface[3].MovementDone) ) THEN
	fbFreeTransport[initax](AxisNo := initax, RequestPosition := WaitingAbsPosition,execute := TRUE);
	IF fbFreeTransport[3].done THEN
	autoexecute := TRUE;
	initdone := TRUE;
	END_IF
END_IF

		FOR i := 1 TO grpcnt DO
			IF NOT MoverInfo[i].reserved THEN
				IF NOT (MoverInterface[i].Setpos = WaitingAbsPosition) THEN
					fbFreeTransport[i](AxisNo := i, RequestPosition := WaitingAbsPosition,execute := autoexecute);
					
				ELSE
					fbFreeTransport[i](AxisNo := i, RequestPosition := WaitingAbsPosition,execute := FALSE);
					IF NOT MoverInfo[i].reserved	THEN
					AwaitingReservationAxis := i;
					END_IF
					//MoverInfo[i].blocked := TRUE;
				END_IF
			
					
			END_IF
		 
		END_FOR

END_FUNCTION_BLOCK

// ---- POUs/CAHandle/FB_CAHandle.TcPOU

FUNCTION_BLOCK FB_CAHandle
VAR_OUTPUT
	initdone: BOOL;
	cadone: BOOL;
	reset: BOOL;
END_VAR
VAR
	state: INT := -10;
	resetstate: INT := 2;
	nextstate: INT;
	halt: BOOL;
	forcedisable: BOOL;
	fbpowerall: FB_PowerAll;
	fbresetall: FB_ResetAll;
	fbaddall: FB_AddAllAxes;
	fbremoveall: FB_RemoveAllAxesCA;
	fbhaltall: FB_HaltAll;
	fbCAgrpEnable: MC_GroupEnableCA(calltargetOID);
	fbCAgrpDisable: MC_GroupDisableCA(calltargetOID);
	fbCAgrpReset: MC_GroupResetCA(calltargetOID);
	fbCAgrpStatus: MC_GroupReadStatusCA;
	fbCAgrpError: MC_GroupReadErrorCA;
	fbuncoupleall: FB_UncoupleAll;
	fbCaInterfaceHandle: ARRAY[1..grpcnt] OF FB_CAInterfaceHandle;
	fbCoupleInit: FB_CoupleInit;
	i: UINT;
	targetpos: ARRAY[1..grpcnt] OF LREAL;
	///targetposact: ARRAY[1..grpcnt] OF LREAL;
	movervel: LREAL := 1000;
	railLength: LREAL := 4000;
END_VAR
VAR_INPUT
	executereset: BOOL := TRUE;
	goon: BOOL;
END_VAR


fbpowerall(enable:=TRUE, axes := poweredaxes);
fbCAgrpStatus(AxesGroup:=CAgrp, enable:=TRUE);
fbCAgrpError(AxesGroup:=CAgrp, enable:=TRUE);

IF (fbpowerall.ison ) AND NOT executereset THEN
	CASE state OF
		
		-10: fbCoupleInit(execute := TRUE,startline := WaitingAbsPosition - 100.0 + ax[1].NcToPlc.moduloactturns * 4000);
			IF fbCoupleInit.done THEN
				state := -5;
			END_IF
			
		-5:	fbaddall(Execute:=FALSE);
			fbaddall(Execute:=TRUE);
			
			(* CAinterface.MoverInterface[1].Targetpos := 1000;
			CAinterface.MoverInterface[2].Targetpos := 1500;
			CAinterface.MoverInterface[3].Targetpos := 2000;
			CAinterface.MoverInterface[4].Targetpos := 2500;
			*)
			state := -4;
		-4:	
			fbaddall();
			IF (NOT fbaddall.Busy) THEN
				IF (NOT fbaddall.Error) THEN
					nextstate := -3;
					state := -3; //100
				END_IF
			END_IF
		-3:
			fbCAgrpEnable(AxesGroup:=CAgrp, execute:=FALSE);
			fbCAgrpEnable(AxesGroup:=CAgrp, execute:=TRUE);
			state := -2;
		-2:
			fbCAgrpEnable(AxesGroup:=CAgrp);
			IF (fbCAgrpEnable.Done) THEN
				ADSLOGSTR(ADSLOG_MSGTYPE_HINT, 'XTS Successfully Activated', '');
				nextstate := 0;
				cadone		:= TRUE;
				state := 0;
			END_IF
		0:	// now all axes are in the enabled group, we start with some moves
			FOR i := 1 TO grpcnt DO
			fbCaInterfaceHandle[i](axisno := i, movervel := MoverInterface[i].Velocity, moveracc := MoverInterface[i].Acceleration);	
			END_FOR	
			initdone := TRUE;
			
			
		5:
			fbhaltall(execute:=FALSE);
			fbhaltall(execute:=TRUE);
			state := 6;
		6:	fbhaltall();
			IF (fbhaltall.Done) THEN
				state := 100;
			END_IF
		10:
			fbCAgrpDisable(AxesGroup:=CAgrp, execute:=FALSE);
			fbCAgrpDisable(AxesGroup:=CAgrp, execute:=TRUE);
			state := 11;
		11:	fbCAgrpDisable(AxesGroup:=CAgrp);
			IF (fbCAgrpDisable.Done) THEN
				state := 12;
			END_IF
		12:
			fbremoveall(Execute:=FALSE);
			fbremoveall(Execute:=TRUE);
			state := 13;
		13:	fbremoveall();
			IF (NOT fbremoveall.Busy) THEN
				IF (NOT fbremoveall.Error) THEN
					ADSLOGSTR(ADSLOG_MSGTYPE_HINT, 'All Axes Removed From Group', '');
					nextstate := 14;
					state := 100;
				END_IF
			END_IF
			
		14:	fbresetall(execute:=FALSE);
			fbresetall(execute:=TRUE);
			state := 15;
		15:
			fbresetall();
			IF (NOT fbresetall.Busy) THEN
				IF (NOT fbresetall.Error) THEN
					ADSLOGSTR(ADSLOG_MSGTYPE_HINT, 'All Axes Successfully Reset', '');
					nextstate := -5;
					state := 100;
				END_IF
			END_IF
			
		16: fbuncoupleall.execute := FALSE;
			state := 17;
		17: fbuncoupleall.execute := TRUE;
			
		100: 
			ADSLOGSTR(ADSLOG_MSGTYPE_HINT, 'Set MAIN.goon to TRUE to continue', '');
			state := 101;
		101:
			IF (goon) THEN				
				state := nextstate;
				goon := FALSE;
			END_IF			

	END_CASE
	
IF (halt) THEN
		state := 5;
		halt := FALSE;
	END_IF
IF (forcedisable) THEN
		state := 10;
		forcedisable := FALSE;
	END_IF
END_IF



FOR i:=1 TO grpcnt DO
	CAInterface.MoverInterface[i].Setpos := GVL.ax[2*i].NcToPlc.ModuloSetPos ;
	IF (ABS(CAInterface.MoverInterface[i].Targetpos - GVL.ax[2*i].NcToPlc.ModuloSetPos)) < 0.1 THEN
		CAInterface.MoverInterface[i].Setpos := CAInterface.MoverInterface[i].Targetpos;
		IF NOT CAInterface.MoverInterface[i].Buddyenable THEN
		CAInterface.MoverInterface[i].MovementDone := TRUE;
		END_IF
	END_IF
	
END_FOR

IF  executereset THEN
	CASE resetstate OF
			
		0: 	FOR i := 1 TO axcnt DO
			poweredaxes[i] := TRUE;
			END_FOR
			resetstate := 2;
		2:	fbuncoupleall.execute := FALSE;
			fbuncoupleall.execute := TRUE;
			resetstate := 3;
		3:	fbuncoupleall();
			IF fbuncoupleall.done OR NOT fbuncoupleall.busy THEN
				resetstate := 4;
			END_IF
		4:	fbCAgrpReset(AxesGroup:=CAgrp, execute:=FALSE);			
			fbCAgrpReset(AxesGroup:=CAgrp, execute:=TRUE);
			resetstate := 5;
		5:  fbCAgrpReset(AxesGroup:=CAgrp);
			IF fbCAgrpReset.Done THEN
				resetstate := 6;
				
			END_IF
		6: 
			fbresetall(execute := FALSE);
			fbresetall(execute := TRUE);
			resetstate := 7;
		7:  
			fbresetall();
			IF NOT fbresetall.busy THEN
				resetstate := 8;
				
			END_IF
		8: 
			fbCAgrpDisable(AxesGroup := CAgrp,Execute := FALSE);
			fbCAgrpDisable(AxesGroup := CAgrp,Execute := TRUE);
			resetstate := 9;
			
		9: fbCAgrpDisable(AxesGroup := CAgrp);
			IF fbCAgrpDisable.Done THEN
				resetstate := 10;
				
			END_IF
		10: fbremoveall.execute := FALSE;
			fbremoveall.execute := TRUE;
			fbremoveall();
			resetstate := 11;
			
		11:  fbremoveall();
			IF fbremoveall.done THEN
				resetstate := 12;
				fbremoveall.execute := FALSE;
			END_IF
		12:
			resetstate := 0;
			executereset := FALSE;
			state := -10;
	END_CASE
ELSE
	resetstate := 0;
END_IF

END_FUNCTION_BLOCK

// ---- POUs/CAHandle/FB_ResetAll.TcPOU
FUNCTION_BLOCK FB_ResetAll
VAR_INPUT
	execute: BOOL;
END_VAR
VAR_OUTPUT
	done: BOOL;
	busy: BOOL;
	error: BOOL;
END_VAR
VAR
	fbreset: ARRAY[1..axcnt] OF MC_Reset;
	fbgrpreset: ARRAY[1..grpcnt] OF MC_Reset;
	i: UINT;
END_VAR


done := TRUE;
busy := FALSE;
error := FALSE;

FOR i:=1 TO axcnt DO
	fbreset[i](Axis:=ax[i], Execute := execute);

	IF (NOT fbreset[i].done) THEN
		done := FALSE;
	END_IF
	IF (fbreset[i].busy) THEN
		busy := TRUE;
	END_IF
	IF (fbreset[i].Error) THEN
		error := TRUE;
	END_IF
END_FOR
FOR i:=1 TO grpcnt DO
	fbgrpreset[i](Axis:=grp[i], Execute := execute);

	IF (NOT fbgrpreset[i].done) THEN
		done := FALSE;
	END_IF
	IF (fbgrpreset[i].busy) THEN
		busy := TRUE;
	END_IF
	IF (fbgrpreset[i].Error) THEN
		error := TRUE;
	END_IF
END_FOR

END_FUNCTION_BLOCK

// ---- POUs/CAHandle/FB_AddAllAxes.TcPOU
FUNCTION_BLOCK FB_AddAllAxes
VAR_INPUT
	execute: BOOL;
END_VAR
VAR_OUTPUT
	done: BOOL;
	busy: BOOL;
	error: BOOL;
END_VAR
VAR
	fbaddtoaxis: ARRAY[1..grpcnt] OF MC_AddAxisToGroupCA(calltargetOID);
	i: UINT;
END_VAR


done := TRUE;
busy := FALSE;
error := FALSE;

FOR i:=1 TO grpcnt DO
	fbaddtoaxis[i](AxesGroup:=CAgrp, Axis :=grp[i], Execute := execute, IdentInGroup := i-1);

	IF (NOT fbaddtoaxis[i].done) THEN
		done := FALSE;
	END_IF
	IF (fbaddtoaxis[i].busy) THEN
		busy := TRUE;
	END_IF
	IF (fbaddtoaxis[i].Error) THEN
		error := TRUE;
	END_IF
END_FOR

END_FUNCTION_BLOCK

// ---- POUs/CAHandle/FB_RemoveAllAxesCA.TcPOU
FUNCTION_BLOCK FB_RemoveAllAxesCA
VAR_INPUT
	execute: BOOL;
END_VAR
VAR_OUTPUT
	done: BOOL;
	busy: BOOL;
	error: BOOL;
END_VAR
VAR
	fbremfromaxis: ARRAY[1..axcnt] OF MC_RemoveAxisFromGroupCA(calltargetOID);
	i: UINT;
END_VAR


done := TRUE;
busy := FALSE;
error := FALSE;

FOR i:=1 TO grpcnt DO
	fbremfromaxis[i](AxesGroup:=CAgrp, Execute := execute, IdentInGroup := i-1);

	IF (NOT fbremfromaxis[i].done) THEN
		done := FALSE;
	END_IF
	IF (fbremfromaxis[i].busy) THEN
		busy := TRUE;
	END_IF
	IF (fbremfromaxis[i].Error) THEN
		error := TRUE;
	END_IF
END_FOR

END_FUNCTION_BLOCK

// ---- POUs/CAHandle/FB_HaltAll.TcPOU
FUNCTION_BLOCK FB_HaltAll
VAR_INPUT
	execute: BOOL;
END_VAR
VAR_OUTPUT
	done: BOOL;
	busy: BOOL;
	error: BOOL;
END_VAR
VAR
	fbhalt: ARRAY[1..grpcnt] OF MC_HaltCA(calltargetOID);
	i: UINT;
END_VAR


done := TRUE;
busy := FALSE;
error := FALSE;

FOR i:=1 TO grpcnt DO
	fbhalt[i](Axis := grp[i], Execute := execute);

	IF (NOT fbhalt[i].done) THEN
		done := FALSE;
	END_IF
	IF (fbhalt[i].busy) THEN
		busy := TRUE;
	END_IF
	IF (fbhalt[i].Error) THEN
		error := TRUE;
	END_IF
END_FOR

END_FUNCTION_BLOCK

// ---- POUs/CAHandle/FB_UncoupleAll.TcPOU
FUNCTION_BLOCK FB_UncoupleAll
VAR_INPUT
	execute: BOOL;
END_VAR
VAR_OUTPUT
	done: BOOL;
	busy: BOOL;
	error: BOOL;
END_VAR
VAR
	fbuncouple: ARRAY[1..axcnt] OF MC_GearOut;
	i: UINT;
END_VAR

done := TRUE;
busy := FALSE;
error := FALSE;
FOR i:=1 TO axcnt DO
	fbuncouple[i](
	Slave:= ax[i], 
	Execute:= execute, 
	Options:= , 
	Done=> , 
	Busy=> , 
	Error=> , 
	ErrorID=> );

	IF (NOT fbuncouple[i].done) THEN
		done := FALSE;
	END_IF
	IF (fbuncouple[i].busy) THEN
		busy := TRUE;
	END_IF
	IF (fbuncouple[i].Error) THEN
		error := TRUE;
	END_IF
END_FOR

END_FUNCTION_BLOCK

// ---- POUs/CAHandle/FB_CAInterfaceHandle.TcPOU
FUNCTION_BLOCK FB_CAInterfaceHandle
VAR_INPUT
	moveracc: LREAL;
	movervel: LREAL;
	axisno: INT;
END_VAR
VAR
	///FBs
	fbhaltsingle: MC_HaltCA(calltargetOID);
	fbmove: MC_MoveAbsoluteCA(calltargetOID);
	buffermode: MC_BufferMode;
	fbBuddyenable: FB_Buddyenable;
	fbBuddyGearBack: FB_BuddygearBack;
	reltargetpos: LREAL;
	targetpos: LREAL;
	acttargetpos: LREAL;
	actclockwise: BOOL;
	buddytemp: BOOL;
	fbSectionChange	: FB_SectionChange;
	///lokal
	state		: INT := 0;
	flip		: BOOL;
	secondcurve	: INT;
END_VAR


CASE state OF 
            	
					0: 	//überprüfen ob änderung
						IF (NOT (acttargetpos = CAinterface.MoverInterface[axisno].Targetpos) )THEN 
							state := 5;
							CAinterface.MoverInterface[axisno].movementdone := FALSE;
						ELSE
							IF NOT(CAinterface.MoverInterface[axisno].Buddyenable=CAinterface.MoverInterface[axisno].Buddyactive)THEN
								state := 13;
							END_IF
						END_IF
					5:	//berechnung
						IF CAinterface.MoverInterface[axisno].Clockwise THEN
							//CLOCKWISE
								IF  (CAinterface.MoverInterface[axisno].Targetpos <ax[2*axisno].NcToPlc.ModuloSetPos) THEN
									reltargetpos := CAinterface.MoverInterface[axisno].Targetpos +  railLength;
								ELSE
									reltargetpos := CAinterface.MoverInterface[axisno].Targetpos;
								END_IF								
							
						ELSE
							//Counter_Clockwise
							IF  (CAinterface.MoverInterface[axisno].Targetpos >ax[2*axisno].NcToPlc.ModuloSetPos) THEN
									reltargetpos := CAinterface.MoverInterface[axisno].Targetpos -  railLength;
							ELSE
									reltargetpos := CAinterface.MoverInterface[axisno].Targetpos;
							END_IF
													
						END_IF
						
						targetpos := reltargetpos +ax[2*axisno].NcToPlc.ModuloSetTurns*raillength;
	
						
            			
						
						 state := 9;
						 acttargetpos := CAinterface.MoverInterface[axisno].Targetpos;
						 actclockwise := CAinterface.MoverInterface[axisno].Clockwise;
						
					9:	fbmove(axis:=grp[axisno], execute:=FALSE);
           		   		fbmove(axis:=grp[axisno], execute:=TRUE, position:=targetpos, velocity:= movervel(*für gläsertest, sonst: movervel*), gap:=CAGap, Acceleration := , ContinuousUpdate := TRUE);///moveracc);
						state := 10;
				
					10:
						fbmove(axis:=grp[axisno]);
						
						//Kurvenscheibe:
						(*
						IF F_MoverInCurve( ax[2*axisno].NcToPlc.ModuloActPos) THEN
							//Auf Änderung der Phase Triggern:
							IF  ax[2*axisno].NcToPlc.ModuloActPos > 1000 AND  ax[2*axisno].NcToPlc.ModuloActPos < 2500 THEN
								secondcurve := 0;
							ELSE
								secondcurve := 1;
							END_IF
							
							fbSectionChange(Position :=secondcurve * raillength+ ax[2*axisno].NcToPlc.ModuloActPos, Clockwise := actclockwise);
							
							// Geschwindigkeit neu setzen;
							fbMove.Velocity := GVL.CurveVelo[fbSectionChange.Phase];
							
							//Execute aus fbSectionchange weitergeben/triggern
							fbmove.Execute := fbSectionChange.Trigger;
						ELSE
							//steigende Flanke auf alte geschwindigkeit	
							IF NOT (fbmove.Velocity = movervel) THEN
								fbmove(axis:=grp[axisno], Velocity := movervel, execute := FALSE);
								fbmove(axis:=grp[axisno], Velocity := movervel, execute := TRUE);
							END_IF
						END_IF
						
						*)
						
						//CAInterface.MoverInterface[axisno].MovementDone := FALSE;
						//unterwegs neue position:
						IF (NOT (acttargetpos = CAinterface.MoverInterface[axisno].Targetpos)) OR (NOT (actclockwise = CAinterface.MoverInterface[axisno].Clockwise)) THEN
							state := 0;
							//state := 20;
							
						END_IF
						
						IF (fbmove.Done AND ((ax[2*axisno].NcToPlc.ModuloSetPos - MoverInterface[axisno].Targetpos)<0.01)) THEN
							IF CAinterface.MoverInterface[axisno].Buddyenable THEN
								
								state := 13;
								fbBuddyenable(execute := FALSE);
								fbBuddyGearBack(execute := FALSE);
								ADSLOGSTR(ADSLOG_MSGTYPE_HINT, 'start uncouple and relative movement', '');
								
							ELSE
							
							state := 0;
							CAInterface.MoverInterface[axisno].MovementDone := TRUE;
							END_IF
						END_IF
						
						
						
						
						
						
					
					13: IF  NOT CAinterface.MoverInterface[axisno].Buddyenable AND fbBuddyenable.done OR mi5.ResetXTS(*!!!!unschoen!!!!*)//OR ( NOT (acttargetpos = CAinterface.MoverInterface[axisno].Targetpos) AND fbBuddyenable.done)
						THEN
						state := 15;
						
						ELSE
							fbBuddyenable(
								execute:= TRUE, 
								axno:= axisno, 
								gap:= CAinterface.MoverInterface[axisno].Buddygap, 
								done=> , 
								);
						IF fbBuddyenable.done  THEN
							state := 14;
							CAinterface.MoverInterface[axisno].Buddyactive := TRUE;
							CAInterface.MoverInterface[axisno].MovementDone := TRUE; ///
						END_IF
						END_IF
						
					14: 
						IF NOT CAinterface.MoverInterface[axisno].Buddyenable OR mi5.ResetXTS THEN
						state := 15;	
						END_IF
						
					
					15: IF  NOT CAinterface.MoverInterface[axisno].Buddyenable THEN
							fbBuddyGearBack(execute := TRUE, axno:= axisno, masterpos := fbBuddyenable.masterpos, slavepos := fbBuddyenable.slavepos);							

						END_IF
						IF fbBuddyGearBack.done THEN
							CAinterface.MoverInterface[axisno].Buddyactive := FALSE;
							state := 0;
							
						END_IF
						
					
						
					20:
						fbhaltsingle(Axis :=grp[axisno],execute:=FALSE);
						fbhaltsingle(execute:=TRUE,Axis :=grp[axisno]);
						state := 21;
					21:	
						fbhaltsingle(Axis :=grp[axisno]);
						IF (fbhaltsingle.Done) THEN
							state := 0;
						END_IF
				END_CASE

END_FUNCTION_BLOCK

// ---- POUs/CAHandle/FB_Buddyenable.TcPOU
FUNCTION_BLOCK FB_Buddyenable
VAR_INPUT
	execute: BOOL;
	axno: INT;
	gap: LREAL;
END_VAR
VAR_OUTPUT
	done: BOOL;
	busy: BOOL;
	masterpos: LREAL;
	slavepos: LREAL;
END_VAR
VAR
	fbMoveAbs: Tc2_MC2.MC_MoveAbsolute;
	fbCouple: Tc2_MC2.MC_GearIn;
	fbDeCouple: Tc2_MC2.MC_GearOut;
	fbDeCoupleCA: Tc2_MC2.MC_GearOut;
	state: INT;
	targetpos: LREAL;
END_VAR

IF Execute THEN
		done 		:= FALSE;
		busy 		:= TRUE;
		CASE state OF
			0:	masterpos   := ax[2*axno].NcToPlc.Setpos;
				slavepos    := ax[2*axno].NcToPlc.Setpos -  couplegap;
				state := 1999;
				IF NOT ((masterpos-slavepos) = couplegap) THEN
					state := 999;
				END_IF
				fbDeCouple(
							Slave:= ax[2*axno-1], 
							Execute:= FALSE, 
							Options:= , 
							Done=> , 
							Busy=> , 
							Error=> , 
							ErrorID=> );
				fbDeCoupleCA(
							Slave:= ax[2*axno], 
							Execute:= FALSE, 
							Options:= , 
							Done=> , 
							Busy=> , 
							Error=> , 
							ErrorID=> );
				state := 2;
			
			2: fbDeCouple(
							Slave:= ax[2*axno-1], 
							Execute:= TRUE, 
							Options:= , 
							Done=> , 
							Busy=> , 
							Error=> , 
							ErrorID=> );
				fbDeCoupleCA(
							Slave:= ax[2*axno], 
							Execute:= TRUE, 
							Options:= , 
							Done=> , 
							Busy=> , 
							Error=> , 
							ErrorID=> );
				IF fbDeCouple.Done AND fbDeCoupleCA.Done THEN 
					state := 3;
				END_IF
			
			3: // Position Berechnen
				targetpos := ax[2*axno].NcToPlc.SetPos - gap;
				fbMoveAbs(	Axis:= ax[2*axno-1], 
							Execute:= FALSE, 							 
							Velocity:= buddyvelo);
				state := 4;
				
			4:	fbMoveAbs(	Axis:= ax[2*axno-1],Position := targetpos, 
							Execute:= TRUE);
				IF (* fbMoveAbs.Done AND *) ax[2*axno-1].NcToPlc.SetPos = targetpos THEN
					
					
					state 		:= 5;
				END_IF
				IF fbMoveAbs.Error THEN
					state := 3;
				END_IF
			
				
				
			5: //
				//GVL.poweredaxes[2*axno-1] := FALSE;
				//GVL.poweredaxes[2*axno] := FALSE;
				
			
			
				
				execute 	:= FALSE;
				done 		:= TRUE;
				state 		:= 0;
			
			
		END_CASE
ELSE
state := 0;
done := FALSE;		
END_IF

END_FUNCTION_BLOCK

// ---- POUs/CAHandle/FB_BuddygearBack.TcPOU
FUNCTION_BLOCK FB_BuddygearBack
VAR_INPUT
	execute: BOOL;
	activate: BOOL;
	release: BOOL;
	axno: INT;
	gap: LREAL;
	masterpos: LREAL;
	slavepos: LREAL;
END_VAR
VAR_OUTPUT
	buddyactive: BOOL;
	buddysafe: BOOL;
	done: BOOL;
	busy: BOOL;
END_VAR
VAR
	powerslave: MC_Power;
	powermaster: MC_Power;
	fbMoveAbsSlave: Tc2_MC2.MC_MoveAbsolute;
	fbMoveAbsMaster: Tc2_MC2.MC_MoveAbsolute;
	fbCouple: Tc2_MC2.MC_GearIn;
	fbCoupleCA: Tc2_MC2.MC_GearIn;
	fbDeCouple: Tc2_MC2.MC_GearOut;
	state: INT;
	targetpos: LREAL;
END_VAR

IF Execute THEN
		busy		:= TRUE;
		done		:= FALSE;
			CASE state OF
			
			0:	
				
			// Position Berechnen
				targetpos := masterpos - couplegap;
				powerslave(Axis := ax[2*axno], Enable := TRUE, Enable_Positive := TRUE, Enable_Negative := TRUE);
				powermaster(Axis := ax[2*axno-1], Enable := TRUE, Enable_Positive := TRUE, Enable_Negative := TRUE);
 				//GVL.poweredaxes[2*axno-1] := TRUE;
				//GVL.poweredaxes[2*axno] := TRUE;
				IF powerslave.Status AND powermaster.Status THEN
					state := 3;
				END_IF
			3:	
				fbMoveAbsMaster(	Axis:= ax[2*axno], 
							Execute:= FALSE, 
							Position:= masterpos, 
							Velocity:= buddyvelo);
				fbMoveAbsSlave(	Axis:= ax[2*axno-1], 
							Execute:= FALSE, 
							Position:= slavepos, 
							Velocity:= buddyvelo);
				state := 10;
				
			10:
				fbMoveAbsMaster(	Axis:= ax[2*axno], 
							Execute:= TRUE);
				
					
				fbMoveAbsSlave(	Axis:= ax[2*axno-1], 
							Execute:= TRUE);
				IF fbMoveAbsMaster.Done AND fbMoveAbsSlave.Done THEN
					state := 20;
				END_IF
				
			20:
				fbCouple(
						Master:= ax[2*axno], 
						Slave:= ax[2*axno -1], 
						Execute:= FALSE 
						);
				fbCoupleCA(
						Master := grp[axno],
						Slave := ax[2*axno],
						execute := FALSE);
				
				state := 30;
			30: fbCouple(
						Master:= ax[2*axno], 
						Slave:= ax[2*axno -1], 
						Execute:= TRUE 
						);
						
				fbCoupleCA(
						Master := grp[axno],
						Slave := ax[2*axno],
						execute := TRUE);
						
						
				IF fbCouple.InGear AND fbCoupleCA.InGear THEN
					state := 40;
				END_IF
			40: 
				buddysafe 	:= TRUE;
				execute		:= FALSE;
				busy		:= FALSE;
				execute		:= TRUE;
				done		:= TRUE;
				state 		:= 0;
			END_CASE		
ELSE
	state := 0;
	done := FALSE;
END_IF

END_FUNCTION_BLOCK

// ---- POUs/CAHandle/MC2Handle/FB_SectionChange.TcPOU
FUNCTION_BLOCK FB_SectionChange
VAR_INPUT
	Position	: LREAL;
	Clockwise	: BOOL;
END_VAR
VAR_OUTPUT
	Phase			: INT;
	Trigger			: BOOL;
END_VAR
VAR
	PhaseMemo	: INT;
	i 	: INT;
END_VAR

FOR i := 1 TO curvesectioncnt DO
	Trigger := TRUE;
	IF ( Position > GVL.CurveSection[i-1]) AND ( Position <= GVL.CurveSection[i] ) THEN
		
		
		IF NOT (Phase = PhaseMemo) THEN
			Trigger := FALSE;
			PhaseMemo := Phase;
		END_IF
		Phase := i + BOOL_TO_INT (clockwise);
	END_IF
END_FOR

END_FUNCTION_BLOCK

// ---- POUs/CAHandle/MC2Handle/FB_CoupleInit.TcPOU
FUNCTION_BLOCK FB_CoupleInit
VAR_INPUT
	execute: BOOL;
	startline: LREAL;
END_VAR
VAR_OUTPUT
	busy: BOOL;
	error: BOOL;
	done: BOOL;
END_VAR
VAR
	fbmoveAbsMC: ARRAY[1..axcnt] OF MC_MoveAbsolute;
	fbcouple: ARRAY[1..grpcnt] OF Tc2_MC2.MC_GearIn;
	fbcoupleCA: ARRAY[1..grpcnt] OF Tc2_MC2.MC_GearIn;
	fbSetpos: ARRAY[1..grpcnt] OF Tc2_MC2.MC_SetPosition;
	state: INT := 0;
	i: INT;
	movedone: BOOL;
	mccoupledone: BOOL;
	CAcoupledone: BOOL;
	setposdone: BOOL;
END_VAR

busy := FALSE;
IF execute THEN
	busy := TRUE;
	done := FALSE;
	CASE state OF
		
	0:	
		startposition[6] := startline;
		startposition[5] := startline - couplegap;
		startposition[4] := startline - 2* couplegap -50;
		startposition[3] := startline - 3* couplegap -50;
		startposition[2] := startline - 4* couplegap -100;
		startposition[1] := startline - 5* couplegap -100;
		
		state := 1;
	1: 
		FOR i := 1 TO axcnt DO
		fbmoveAbsMC[i](Axis := ax[i],Position := Startposition[i], Velocity := 400, Execute := FALSE);
		END_FOR
		state := 2;
		
	2:	
		movedone := TRUE;
		FOR i := 1 TO axcnt DO
			fbmoveAbsMC[i](Axis := ax[i],Position := Startposition[i], Velocity := 400, Execute := TRUE);
			IF NOT fbmoveAbsMC[i].Done THEN movedone := FALSE; END_IF
		END_FOR
		IF movedone THEN
			state := 9;
		END_IF
		
	9:	//MC2 couplen
		FOR i := 1 TO grpcnt DO
		fbcouple[i](Master := ax[2*i], Slave := ax[2*i-1],execute := FALSE); 
		END_FOR
		state := 10;
		
	10: //MC2 couplen
		mccoupledone := TRUE;
			FOR i := 1 TO grpcnt DO
			fbcouple[i](Master := ax[2*i], Slave := ax[2*i-1], execute := TRUE); 
			IF fbcouple[i].Busy THEN
				mccoupledone := FALSE;
			END_IF	
		END_FOR
		IF mccoupledone THEN state := 15; END_IF


	15: //	setpos virtuelle ca mover
		setposdone := FALSE;
		FOR i := 1 TO grpcnt DO
		fbSetpos[i](Axis := grp[i], Position := ax[2*i].NcToPlc.SetPos,execute := FALSE);
		END_FOR
		state := 16;
		
	16: 
		setposdone := TRUE;
		FOR i := 1 TO grpcnt DO
			fbSetpos[i](Axis := grp[i], Position := ax[2*i].NcToPlc.SetPos,execute := TRUE);
			IF fbSetpos[i].Busy THEN
				setposdone := FALSE;
			END_IF
		END_FOR
		IF setposdone THEN
			state := 20;
		END_IF
		
	20:	// CA couplen
		FOR i := 1 TO grpcnt DO
		fbcoupleCA[i](Master := Grp[i], Slave := ax[2*i],execute := FALSE); 
		END_FOR
		state := 21;
		
	21:
		CAcoupledone := TRUE;
			FOR i := 1 TO grpcnt DO
			fbcoupleCA[i](Master := Grp[i], Slave := ax[2*i],execute := TRUE); 
			IF fbcoupleCA[i].Busy THEN
				CAcoupledone := FALSE;
			END_IF	
		END_FOR
		IF CAcoupledone THEN state := 100; END_IF
		
		
	100: // done
		done 	:= TRUE;
		busy 	:= FALSE;
		execute := FALSE;
		state 	:= 0;
		error := FALSE;
		

	END_CASE

END_IF

END_FUNCTION_BLOCK

// ---- POUs/SkillHandle/VisuLampen/FB_SimuLampHandle.TcPOU
FUNCTION_BLOCK FB_SimuLampHandle
VAR_INPUT
	execute: BOOL;
END_VAR
VAR_OUTPUT
END_VAR
VAR
	fbCheckLamp	: ARRAY[1..ColourCnt] OF ARRAY [1..LampCnt] OF FB_CheckSimuVisu;
	i : INT;
	j : INT;
	LampWith	: LREAL;
	Timer		: ARRAY [1..GrpCnt] OF TOF;
	Blinker		: ARRAY [1..GrpCnt] OF TON;
	RTrigger		: ARRAY [1..GrpCnt] OF R_TRIG;
	FTrigger		: ARRAY [1..GrpCnt] OF F_TRIG;
	changedetected	: ARRAY [1..GrpCnt] OF BOOL;
	blink		: ARRAY [1..GrpCNt] OF BOOL;
END_VAR

LampWith := raillength/LampCnt;
IF execute THEN
	

	FOR i := 1 TO grpcnt DO
		
		RTrigger[i](CLK := MoverInfo[i].reserved);
		FTrigger[i](CLK := MoverInfo[i].reserved);
		IF RTrigger[i].Q OR fTrigger[i].Q THEN
			changedetected[i] := TRUE;
			Timer[i](IN := TRUE);
		END_IF
		IF changedetected[i] THEN
			Timer[i](IN := FALSE, PT := T#1S);
			changedetected[i] := Timer[i].Q;
			Blinker[i](IN := TRUE, PT := T#0.2S);
			IF BLinker[i].Q THEN
				BLinker[i](IN := FALSE);
				blink[i] := NOT blink[i];
			END_IF
		ELSE
			blink[i] := TRUE;
		END_IF
		
		FOR j := 1 TO LampCnt DO
			
			fbCheckLamp[i][j](LampPosition := j*LampWith + 0.5 * LampWith + 20, CheckMoverNo := i, Execute := TRUE, Lamp => LampInterface[i][j]);
			IF NOT blink[i] THEN 
			LampInterface[i][j] := FALSE;
				
			END_IF
		END_FOR
	
	
	END_FOR

END_IF

END_FUNCTION_BLOCK

// ---- POUs/SkillHandle/VisuLampen/FB_CheckSimuVisu.TcPOU
FUNCTION_BLOCK FB_CheckSimuVisu
VAR_INPUT
	LampPosition: LREAL;
	CheckMoverNo: INT;
	Execute: BOOL;
END_VAR
VAR_OUTPUT
	Lamp	: BOOL;
	
END_VAR
VAR
	
END_VAR

IF Execute THEN
	LAMP := FALSE;
		IF MoverInfo[CheckMoverNo].postposition>MoverInfo[CheckMoverNo].preposition 
		THEN
				//DER RESERVIERTE BEREICH GEHT NICHT ÜBER NULL:	
					
					// gesamter bereich umschlungen?
					IF LampPosition >  MoverInfo[CheckMoverNo].preposition AND LampPosition <= MoverInfo[CheckMoverNo].PostPosition THEN
						Lamp:= TRUE;
					END_IF
				
				ELSE
				//DER RESERVIERTE BEREICH GEHT ÜBER NULL!
				//Bereich 1: 0 bis Postpos:
					// Grenze in Bereich?
					IF((LampPosition>=0.0) AND (LampPosition<=MoverInfo[CheckMoverNo].postposition)) 
						THEN 
							Lamp := TRUE;
								
					END_IF
				
				//Bereich 2: Prepos bis 4000
					// Grenze in Bereich?
					IF((LampPosition>=MoverInfo[CheckMoverNo].preposition) AND (LampPosition<=raillength)) 
						THEN 
							Lamp := TRUE;
					END_IF	
		END_IF
				
END_IF

END_FUNCTION_BLOCK

// ---- POUs/FB_TranslateInterface.TcPOU
FUNCTION_BLOCK FB_TranslateInterface
VAR_INPUT
	execute : BOOL := TRUE;
END_VAR
VAR_OUTPUT
END_VAR
VAR
 mypointer	: POINTER TO DUT_MODULE_INTERFACE_OUTPUT;
 
END_VAR

